# EPICS substitutions: evrMrmApp/Db/evr-pcie-300dc.substitutions
# Record set for a PCIe-EVR-300DC
#
# Macros:
#  EVR = Card name (same as mrmEvrSetupPCI())
#  SYS = System name (ie SR-TM)
#  D = Device name (ie EVR:Diag2)
#  FEVT = Event link frequency (default 124.916 MHz)
#
# Record names have the general forms:
#  $(SYS){$(D)}Signal-SD
#  $(SYS){$(D)-SubDev}Signal-SD

file "mrmevrbase.template"
{
{P="$(SYS){$(D)}", OBJ="$(EVR)", EVNT1HZ="\$(EVNT1HZ=125)", FEVT="\$(FEVT=124.916)"}
}

file "databuftx.db"
{pattern
{P, OBJ, PROTO}
{"$(SYS){$(D)}", "$(EVR):BUFTX", 1}
}

file "evrSoftEvt.template"
{
{P="$(SYS){$(D)}", OBJ="$(EVR)"}
}

file "databuftxCtrl.db"
{pattern
{P, OBJ}
{"$(SYS){$(D)}", "$(EVR):BUFTX"}
}

file "mrmevrbufrx.db"
{pattern
{P, OBJ, PROTO}
{"$(SYS){$(D)}", $(EVR):BUFRX, 0xff00}
}

file mrmSoftSeq.template {
pattern { P, EVG, seqNum, NELM }
{ "$(SYS){$(D)-SoftSeq:0}", $(EVR), 0, 2047 }
{ "$(SYS){$(D)-SoftSeq:1}", $(EVR), 1, 2047 }
{ "$(SYS){$(D)-SoftSeq:2}", $(EVR), 2, 2047 }
}

file evrSoftSeq.template {
pattern { P, EVG, seqNum, NELM }
{ "$(SYS){$(D)-SoftSeq:0}", $(EVR), 0, 2047 }
{ "$(SYS){$(D)-SoftSeq:1}", $(EVR), 1, 2047 }
{ "$(SYS){$(D)-SoftSeq:2}", $(EVR), 2, 2047 }
}

file "sfp.db"
{
{P="$(SYS){$(D)-SFP}", OBJ="$(EVR):SFP"}
}

file "mrmevrdc.template"
{
{P="$(SYS){$(D)-DC}", OBJ="$(EVR)"}
}

file "evrmap.db"
{pattern
{NAME, OBJ, func, EVT}
{"$(SYS){$(D)}Evt:Blink0-SP", "$(EVR)", Blink, 15}
{"$(SYS){$(D)}Evt:Blink1-SP", "$(EVR)", Blink, 0}
{"$(SYS){$(D)}Evt:ResetPS-SP","$(EVR)", "Reset PS", 123}
}

file "evrevent.db"
{pattern
{EN, OBJ, CODE, EVNT}
{"$(SYS){$(D)}1hz",  "$(EVR)", 0x7d, 125}
{"$(SYS){$(D)}EvtA", "$(EVR)", 10, 10}
{"$(SYS){$(D)}EvtB", "$(EVR)", 11, 11}
{"$(SYS){$(D)}EvtC", "$(EVR)", 12, 12}
{"$(SYS){$(D)}EvtD", "$(EVR)", 13, 13}
{"$(SYS){$(D)}EvtE", "$(EVR)", 14, 14}
{"$(SYS){$(D)}EvtF", "$(EVR)", 15, 15}
{"$(SYS){$(D)}EvtG", "$(EVR)", 16, 16}
{"$(SYS){$(D)}EvtH", "$(EVR)", 17, 17}
}

file "evrscale.db"
{pattern
{IDX, P, SN, OBJ, MAX}
{0, "$(SYS){$(D)}", "$(SYS){$(D)-PS:$(IDX)}", "$(EVR):PS$(IDX)", "0xffffffff"}
{1, "$(SYS){$(D)}", "$(SYS){$(D)-PS:$(IDX)}", "$(EVR):PS$(IDX)", "0xffffffff"}
{2, "$(SYS){$(D)}", "$(SYS){$(D)-PS:$(IDX)}", "$(EVR):PS$(IDX)", "0xffffffff"}
{3, "$(SYS){$(D)}", "$(SYS){$(D)-PS:$(IDX)}", "$(EVR):PS$(IDX)", "0xffffffff"}
{4, "$(SYS){$(D)}", "$(SYS){$(D)-PS:$(IDX)}", "$(EVR):PS$(IDX)", "0xffffffff"}
{5, "$(SYS){$(D)}", "$(SYS){$(D)-PS:$(IDX)}", "$(EVR):PS$(IDX)", "0xffffffff"}
{6, "$(SYS){$(D)}", "$(SYS){$(D)-PS:$(IDX)}", "$(EVR):PS$(IDX)", "0xffffffff"}
{7, "$(SYS){$(D)}", "$(SYS){$(D)-PS:$(IDX)}", "$(EVR):PS$(IDX)", "0xffffffff"}
}

file "mrmevrout.db"
{pattern
{ON, OBJ, DESC}
{"$(SYS){$(D)-Out:Int}", "$(EVR):Int", "Internal"}
# IFB appears in reg map as FPUV, by we name it as RTM
# default to tri-state
pattern
{ON, OBJ, DESC, DEFAULT}
{"$(SYS){$(D)-Out:RB00}", "$(EVR):FrontUnivOut0", "UNIV0", 61}
{"$(SYS){$(D)-Out:RB01}", "$(EVR):FrontUnivOut1", "UNIV1", 61}
{"$(SYS){$(D)-Out:RB02}", "$(EVR):FrontUnivOut2", "UNIV2", 61}
{"$(SYS){$(D)-Out:RB03}", "$(EVR):FrontUnivOut3", "UNIV3", 61}
{"$(SYS){$(D)-Out:RB04}", "$(EVR):FrontUnivOut4", "UNIV4", 61}
{"$(SYS){$(D)-Out:RB05}", "$(EVR):FrontUnivOut5", "UNIV5", 61}
{"$(SYS){$(D)-Out:RB06}", "$(EVR):FrontUnivOut6", "UNIV6", 61}
{"$(SYS){$(D)-Out:RB07}", "$(EVR):FrontUnivOut7", "UNIV7", 61}
{"$(SYS){$(D)-Out:RB08}", "$(EVR):FrontUnivOut8", "UNIV8", 61}
{"$(SYS){$(D)-Out:RB09}", "$(EVR):FrontUnivOut9", "UNIV9", 61}
{"$(SYS){$(D)-Out:RB10}", "$(EVR):FrontUnivOut10", "UNIV10", 61}
{"$(SYS){$(D)-Out:RB11}", "$(EVR):FrontUnivOut11", "UNIV11", 61}
{"$(SYS){$(D)-Out:RB12}", "$(EVR):FrontUnivOut12", "UNIV12", 61}
{"$(SYS){$(D)-Out:RB13}", "$(EVR):FrontUnivOut13", "UNIV13", 61}
{"$(SYS){$(D)-Out:RB14}", "$(EVR):FrontUnivOut14", "UNIV14", 61}
{"$(SYS){$(D)-Out:RB15}", "$(EVR):FrontUnivOut15", "UNIV15", 61}
}

file "mrmevroutint.db"
{{
    ON="$(SYS){$(D)-Out:Int}", OBJ="$(EVR)"
}}

# Pulse generators w/o a prescaler set NOPS=1
file "evrpulser.db"
{pattern
{PID, P, PN, OBJ, DMAX, WMAX, PMAX, NOPS}
{0, "$(SYS){$(D)}", "$(SYS){$(D)-DlyGen:$(PID)}", "$(EVR):Pul$(PID)", "0xffffffff", "0xffffffff", "0xffff", 0}
{1, "$(SYS){$(D)}", "$(SYS){$(D)-DlyGen:$(PID)}", "$(EVR):Pul$(PID)", "0xffffffff", "0xffffffff", "0xffff", 0}
{2, "$(SYS){$(D)}", "$(SYS){$(D)-DlyGen:$(PID)}", "$(EVR):Pul$(PID)", "0xffffffff", "0xffffffff", "0xffff", 0}
{3, "$(SYS){$(D)}", "$(SYS){$(D)-DlyGen:$(PID)}", "$(EVR):Pul$(PID)", "0xffffffff", "0xffffffff", "0xffff", 0}
{4, "$(SYS){$(D)}", "$(SYS){$(D)-DlyGen:$(PID)}", "$(EVR):Pul$(PID)", "0xffffffff", "0xffff", "1", 1}
{5, "$(SYS){$(D)}", "$(SYS){$(D)-DlyGen:$(PID)}", "$(EVR):Pul$(PID)", "0xffffffff", "0xffff", "1", 1}
{6, "$(SYS){$(D)}", "$(SYS){$(D)-DlyGen:$(PID)}", "$(EVR):Pul$(PID)", "0xffffffff", "0xffff", "1", 1}
{7, "$(SYS){$(D)}", "$(SYS){$(D)-DlyGen:$(PID)}", "$(EVR):Pul$(PID)", "0xffffffff", "0xffff", "1", 1}
{8, "$(SYS){$(D)}", "$(SYS){$(D)-DlyGen:$(PID)}", "$(EVR):Pul$(PID)", "0xffffffff", "0xffff", "1", 1}
{9, "$(SYS){$(D)}", "$(SYS){$(D)-DlyGen:$(PID)}", "$(EVR):Pul$(PID)", "0xffffffff", "0xffff", "1", 1}
{10,"$(SYS){$(D)}", "$(SYS){$(D)-DlyGen:$(PID)}", "$(EVR):Pul$(PID)", "0xffffffff", "0xffff", "1", 1}
{11,"$(SYS){$(D)}", "$(SYS){$(D)-DlyGen:$(PID)}", "$(EVR):Pul$(PID)", "0xffffffff", "0xffff", "1", 1}
{12,"$(SYS){$(D)}", "$(SYS){$(D)-DlyGen:$(PID)}", "$(EVR):Pul$(PID)", "0xffffffff", "0xffff", "1", 1}
{13,"$(SYS){$(D)}", "$(SYS){$(D)-DlyGen:$(PID)}", "$(EVR):Pul$(PID)", "0xffffffff", "0xffff", "1", 1}
{14,"$(SYS){$(D)}", "$(SYS){$(D)-DlyGen:$(PID)}", "$(EVR):Pul$(PID)", "0xffffffff", "0xffff", "1", 1}
{15,"$(SYS){$(D)}", "$(SYS){$(D)-DlyGen:$(PID)}", "$(EVR):Pul$(PID)", "0xffffffff", "0xffff", "1", 1}
# gate generators
{28,"$(SYS){$(D)}", "$(SYS){$(D)-DlyGen:$(PID)}", "$(EVR):Pul$(PID)", "0xffffffff", "0xffff", "1", 1}
{29,"$(SYS){$(D)}", "$(SYS){$(D)-DlyGen:$(PID)}", "$(EVR):Pul$(PID)", "0xffffffff", "0xffff", "1", 1}
{30,"$(SYS){$(D)}", "$(SYS){$(D)-DlyGen:$(PID)}", "$(EVR):Pul$(PID)", "0xffffffff", "0xffff", "1", 1}
{31,"$(SYS){$(D)}", "$(SYS){$(D)-DlyGen:$(PID)}", "$(EVR):Pul$(PID)", "0xffffffff", "0xffff", "1", 1}
}

# Default to 3 possible trigger mappings per pulser
file "evrpulsermap.db"
{pattern
{PID, NAME, OBJ, F, EVT}
{0, "$(SYS){$(D)-DlyGen:$(PID)}Evt:Trig0-SP", "$(EVR):Pul$(PID)", Trig, 0}
{0, "$(SYS){$(D)-DlyGen:$(PID)}Evt:Trig1-SP", "$(EVR):Pul$(PID)", Trig, 0}
{0, "$(SYS){$(D)-DlyGen:$(PID)}Evt:Trig2-SP", "$(EVR):Pul$(PID)", Trig, 0}
{1, "$(SYS){$(D)-DlyGen:$(PID)}Evt:Trig0-SP", "$(EVR):Pul$(PID)", Trig, 0}
{1, "$(SYS){$(D)-DlyGen:$(PID)}Evt:Trig1-SP", "$(EVR):Pul$(PID)", Trig, 0}
{1, "$(SYS){$(D)-DlyGen:$(PID)}Evt:Trig2-SP", "$(EVR):Pul$(PID)", Trig, 0}
{2, "$(SYS){$(D)-DlyGen:$(PID)}Evt:Trig0-SP", "$(EVR):Pul$(PID)", Trig, 0}
{2, "$(SYS){$(D)-DlyGen:$(PID)}Evt:Trig1-SP", "$(EVR):Pul$(PID)", Trig, 0}
{2, "$(SYS){$(D)-DlyGen:$(PID)}Evt:Trig2-SP", "$(EVR):Pul$(PID)", Trig, 0}
{3, "$(SYS){$(D)-DlyGen:$(PID)}Evt:Trig0-SP", "$(EVR):Pul$(PID)", Trig, 0}
{3, "$(SYS){$(D)-DlyGen:$(PID)}Evt:Trig1-SP", "$(EVR):Pul$(PID)", Trig, 0}
{3, "$(SYS){$(D)-DlyGen:$(PID)}Evt:Trig2-SP", "$(EVR):Pul$(PID)", Trig, 0}
{4, "$(SYS){$(D)-DlyGen:$(PID)}Evt:Trig0-SP", "$(EVR):Pul$(PID)", Trig, 0}
{4, "$(SYS){$(D)-DlyGen:$(PID)}Evt:Trig1-SP", "$(EVR):Pul$(PID)", Trig, 0}
{4, "$(SYS){$(D)-DlyGen:$(PID)}Evt:Trig2-SP", "$(EVR):Pul$(PID)", Trig, 0}
{5, "$(SYS){$(D)-DlyGen:$(PID)}Evt:Trig0-SP", "$(EVR):Pul$(PID)", Trig, 0}
{5, "$(SYS){$(D)-DlyGen:$(PID)}Evt:Trig1-SP", "$(EVR):Pul$(PID)", Trig, 0}
{5, "$(SYS){$(D)-DlyGen:$(PID)}Evt:Trig2-SP", "$(EVR):Pul$(PID)", Trig, 0}
{6, "$(SYS){$(D)-DlyGen:$(PID)}Evt:Trig0-SP", "$(EVR):Pul$(PID)", Trig, 0}
{6, "$(SYS){$(D)-DlyGen:$(PID)}Evt:Trig1-SP", "$(EVR):Pul$(PID)", Trig, 0}
{6, "$(SYS){$(D)-DlyGen:$(PID)}Evt:Trig2-SP", "$(EVR):Pul$(PID)", Trig, 0}
{7, "$(SYS){$(D)-DlyGen:$(PID)}Evt:Trig0-SP", "$(EVR):Pul$(PID)", Trig, 0}
{7, "$(SYS){$(D)-DlyGen:$(PID)}Evt:Trig1-SP", "$(EVR):Pul$(PID)", Trig, 0}
{7, "$(SYS){$(D)-DlyGen:$(PID)}Evt:Trig2-SP", "$(EVR):Pul$(PID)", Trig, 0}
{8, "$(SYS){$(D)-DlyGen:$(PID)}Evt:Trig0-SP", "$(EVR):Pul$(PID)", Trig, 0}
{8, "$(SYS){$(D)-DlyGen:$(PID)}Evt:Trig1-SP", "$(EVR):Pul$(PID)", Trig, 0}
{8, "$(SYS){$(D)-DlyGen:$(PID)}Evt:Trig2-SP", "$(EVR):Pul$(PID)", Trig, 0}
{9, "$(SYS){$(D)-DlyGen:$(PID)}Evt:Trig0-SP", "$(EVR):Pul$(PID)", Trig, 0}
{9, "$(SYS){$(D)-DlyGen:$(PID)}Evt:Trig1-SP", "$(EVR):Pul$(PID)", Trig, 0}
{9, "$(SYS){$(D)-DlyGen:$(PID)}Evt:Trig2-SP", "$(EVR):Pul$(PID)", Trig, 0}
{10,"$(SYS){$(D)-DlyGen:$(PID)}Evt:Trig0-SP", "$(EVR):Pul$(PID)", Trig, 0}
{10,"$(SYS){$(D)-DlyGen:$(PID)}Evt:Trig1-SP", "$(EVR):Pul$(PID)", Trig, 0}
{10,"$(SYS){$(D)-DlyGen:$(PID)}Evt:Trig2-SP", "$(EVR):Pul$(PID)", Trig, 0}
{11,"$(SYS){$(D)-DlyGen:$(PID)}Evt:Trig0-SP", "$(EVR):Pul$(PID)", Trig, 0}
{11,"$(SYS){$(D)-DlyGen:$(PID)}Evt:Trig1-SP", "$(EVR):Pul$(PID)", Trig, 0}
{11,"$(SYS){$(D)-DlyGen:$(PID)}Evt:Trig2-SP", "$(EVR):Pul$(PID)", Trig, 0}
{12,"$(SYS){$(D)-DlyGen:$(PID)}Evt:Trig0-SP", "$(EVR):Pul$(PID)", Trig, 0}
{12,"$(SYS){$(D)-DlyGen:$(PID)}Evt:Trig1-SP", "$(EVR):Pul$(PID)", Trig, 0}
{12,"$(SYS){$(D)-DlyGen:$(PID)}Evt:Trig2-SP", "$(EVR):Pul$(PID)", Trig, 0}
{13,"$(SYS){$(D)-DlyGen:$(PID)}Evt:Trig0-SP", "$(EVR):Pul$(PID)", Trig, 0}
{13,"$(SYS){$(D)-DlyGen:$(PID)}Evt:Trig1-SP", "$(EVR):Pul$(PID)", Trig, 0}
{13,"$(SYS){$(D)-DlyGen:$(PID)}Evt:Trig2-SP", "$(EVR):Pul$(PID)", Trig, 0}
{14,"$(SYS){$(D)-DlyGen:$(PID)}Evt:Trig0-SP", "$(EVR):Pul$(PID)", Trig, 0}
{14,"$(SYS){$(D)-DlyGen:$(PID)}Evt:Trig1-SP", "$(EVR):Pul$(PID)", Trig, 0}
{14,"$(SYS){$(D)-DlyGen:$(PID)}Evt:Trig2-SP", "$(EVR):Pul$(PID)", Trig, 0}
{15,"$(SYS){$(D)-DlyGen:$(PID)}Evt:Trig0-SP", "$(EVR):Pul$(PID)", Trig, 0}
{15,"$(SYS){$(D)-DlyGen:$(PID)}Evt:Trig1-SP", "$(EVR):Pul$(PID)", Trig, 0}
{15,"$(SYS){$(D)-DlyGen:$(PID)}Evt:Trig2-SP", "$(EVR):Pul$(PID)", Trig, 0}
# gate generators mappings
{28,"$(SYS){$(D)-DlyGen:$(PID)}Evt:Trig0-SP", "$(EVR):Pul$(PID)", Trig, 0}
{28,"$(SYS){$(D)-DlyGen:$(PID)}Evt:Trig1-SP", "$(EVR):Pul$(PID)", Trig, 0}
{28,"$(SYS){$(D)-DlyGen:$(PID)}Evt:Trig2-SP", "$(EVR):Pul$(PID)", Trig, 0}
{29,"$(SYS){$(D)-DlyGen:$(PID)}Evt:Trig0-SP", "$(EVR):Pul$(PID)", Trig, 0}
{29,"$(SYS){$(D)-DlyGen:$(PID)}Evt:Trig1-SP", "$(EVR):Pul$(PID)", Trig, 0}
{29,"$(SYS){$(D)-DlyGen:$(PID)}Evt:Trig2-SP", "$(EVR):Pul$(PID)", Trig, 0}
{30,"$(SYS){$(D)-DlyGen:$(PID)}Evt:Trig0-SP", "$(EVR):Pul$(PID)", Trig, 0}
{30,"$(SYS){$(D)-DlyGen:$(PID)}Evt:Trig1-SP", "$(EVR):Pul$(PID)", Trig, 0}
{30,"$(SYS){$(D)-DlyGen:$(PID)}Evt:Trig2-SP", "$(EVR):Pul$(PID)", Trig, 0}
{31,"$(SYS){$(D)-DlyGen:$(PID)}Evt:Trig0-SP", "$(EVR):Pul$(PID)", Trig, 0}
{31,"$(SYS){$(D)-DlyGen:$(PID)}Evt:Trig1-SP", "$(EVR):Pul$(PID)", Trig, 0}
{31,"$(SYS){$(D)-DlyGen:$(PID)}Evt:Trig2-SP", "$(EVR):Pul$(PID)", Trig, 0}
}

# pulser masking controls
file "evrdcpulser.template"
{pattern
{PID, P, PN, OBJ}
{0, "$(SYS){$(D)}", "$(SYS){$(D)-DlyGen:$(PID)}", "$(EVR):Pul$(PID)"}
{1, "$(SYS){$(D)}", "$(SYS){$(D)-DlyGen:$(PID)}", "$(EVR):Pul$(PID)"}
{2, "$(SYS){$(D)}", "$(SYS){$(D)-DlyGen:$(PID)}", "$(EVR):Pul$(PID)"}
{3, "$(SYS){$(D)}", "$(SYS){$(D)-DlyGen:$(PID)}", "$(EVR):Pul$(PID)"}
{4, "$(SYS){$(D)}", "$(SYS){$(D)-DlyGen:$(PID)}", "$(EVR):Pul$(PID)"}
{5, "$(SYS){$(D)}", "$(SYS){$(D)-DlyGen:$(PID)}", "$(EVR):Pul$(PID)"}
{6, "$(SYS){$(D)}", "$(SYS){$(D)-DlyGen:$(PID)}", "$(EVR):Pul$(PID)"}
{7, "$(SYS){$(D)}", "$(SYS){$(D)-DlyGen:$(PID)}", "$(EVR):Pul$(PID)"}
{8, "$(SYS){$(D)}", "$(SYS){$(D)-DlyGen:$(PID)}", "$(EVR):Pul$(PID)"}
{9, "$(SYS){$(D)}", "$(SYS){$(D)-DlyGen:$(PID)}", "$(EVR):Pul$(PID)"}
{10, "$(SYS){$(D)}", "$(SYS){$(D)-DlyGen:$(PID)}", "$(EVR):Pul$(PID)"}
{11, "$(SYS){$(D)}", "$(SYS){$(D)-DlyGen:$(PID)}", "$(EVR):Pul$(PID)"}
{12, "$(SYS){$(D)}", "$(SYS){$(D)-DlyGen:$(PID)}", "$(EVR):Pul$(PID)"}
{13, "$(SYS){$(D)}", "$(SYS){$(D)-DlyGen:$(PID)}", "$(EVR):Pul$(PID)"}
{14, "$(SYS){$(D)}", "$(SYS){$(D)-DlyGen:$(PID)}", "$(EVR):Pul$(PID)"}
{15, "$(SYS){$(D)}", "$(SYS){$(D)-DlyGen:$(PID)}", "$(EVR):Pul$(PID)"}
}

file "evrin.db"
{pattern
{IN, OBJ, DESC}
# Front panel inputs 4
{"$(SYS){$(D)-In:0}", "$(EVR):FPIn0", "FPIN0 (TTL)"}
{"$(SYS){$(D)-In:1}", "$(EVR):FPIn1", "FPIN1 (TTL)"}
{"$(SYS){$(D)-In:2}", "$(EVR):FPIn2", "FPIN2 (TTL)"}
{"$(SYS){$(D)-In:3}", "$(EVR):FPIn3", "FPIN3 (TTL)"}
# Univ inputs 20
{"$(SYS){$(D)-UnivIn:0}", "$(EVR):FPIn4", "UnivIN0 (TTL)"}
{"$(SYS){$(D)-UnivIn:1}", "$(EVR):FPIn5", "UnivIN1 (TTL)"}
{"$(SYS){$(D)-UnivIn:2}", "$(EVR):FPIn6", "UnivIN2 (TTL)"}
{"$(SYS){$(D)-UnivIn:3}", "$(EVR):FPIn7", "UnivIN3 (TTL)"}
{"$(SYS){$(D)-UnivIn:4}", "$(EVR):FPIn8", "UnivIN4 (TTL)"}
{"$(SYS){$(D)-UnivIn:5}", "$(EVR):FPIn9", "UnivIN5 (TTL)"}
{"$(SYS){$(D)-UnivIn:6}", "$(EVR):FPIn10", "UnivIN6 (TTL)"}
{"$(SYS){$(D)-UnivIn:7}", "$(EVR):FPIn11", "UnivIN7 (TTL)"}
{"$(SYS){$(D)-UnivIn:8}", "$(EVR):FPIn12", "UnivIN8 (TTL)"}
{"$(SYS){$(D)-UnivIn:9}", "$(EVR):FPIn13", "UnivIN9 (TTL)"}
{"$(SYS){$(D)-UnivIn:10}", "$(EVR):FPIn14", "UnivIN10 (TTL)"}
{"$(SYS){$(D)-UnivIn:11}", "$(EVR):FPIn15", "UnivIN11 (TTL)"}
{"$(SYS){$(D)-UnivIn:12}", "$(EVR):FPIn16", "UnivIN12 (TTL)"}
{"$(SYS){$(D)-UnivIn:13}", "$(EVR):FPIn17", "UnivIN13 (TTL)"}
{"$(SYS){$(D)-UnivIn:14}", "$(EVR):FPIn18", "UnivIN14 (TTL)"}
{"$(SYS){$(D)-UnivIn:15}", "$(EVR):FPIn19", "UnivIN15 (TTL)"}
{"$(SYS){$(D)-UnivIn:16}", "$(EVR):FPIn20", "UnivIN16 (TTL)"}
{"$(SYS){$(D)-UnivIn:17}", "$(EVR):FPIn21", "UnivIN17 (TTL)"}
{"$(SYS){$(D)-UnivIn:18}", "$(EVR):FPIn22", "UnivIN18 (TTL)"}
{"$(SYS){$(D)-UnivIn:19}", "$(EVR):FPIn23", "UnivIN19 (TTL)"}
## Backplane inputs 8
}
